Staubli VAL3: typeCenter.pgx

public program typeCenter(num x_nY (dimensions=1), string& x_sStr[] (dimensions=1), num x_nLength (dimensions=1), bool x_bShow (dimensions=1))
  local num lX
  local num lLenStr
  local string lStr
  local num i
begin
  //---------------------------------
  //  S H O W   O N E   S T R I N G
  //---------------------------------
  // type one message in center
  // of the userPage
  //
  // See type()
  //
  lLenStr=getDisplayLen(x_sStr)
  if (lLenStr>x_nLength)
    // comprime
    call strlength(x_sStr,x_nLength)
    lX=(40-x_nLength)/2
  else
    // found the median pos
    lX=20-(lLenStr/2)
    lStr=x_sStr
  endIf
  if x_bShow
    // print on the screen
    call type(lX,x_nY,lStr)
  else
    // add empty space to the string
    for i=1 to lX-1
      lStr=" "+lStr
    endFor
    call strfill(lStr,x_nLength,x_sStr)
  endIf
end
